Fanuc KAREL source: ks00024.KL

-- PROVISIONAL review KL for V770-1; original PC SHA256 53585f96d77963e720301fc55671df62e22ac8339c7abe528639a41481cd47b0
-- Incomplete behavior may be omitted. Consult companion uncertainty JSON. Do not deploy.
PROGRAM KS00024
%NOLOCKGROUP
VAR
  FLAG : BOOLEAN
  N : INTEGER
  STATUS : INTEGER
  PN : STRING[80]
  VN : STRING[80]
-- UNRESOLVED_DECL A type=001101
-- UNRESOLVED_DECL B type=001101
BEGIN
  -- UNRESOLVED_PC offsets 5-13; opcodes 3F,75
  -- UNRESOLVED_PC offsets 18-27; opcodes 3F,75
  -- UNRESOLVED_PC offsets 32-47; opcodes 22,22,30
  -- UNRESOLVED_PC offsets 52-56; opcodes 7F
END KS00024
